SUBAPPLICATION Uebung_001_P (* DigitalInput_I1 auf DigitalOutput_Q1, mit Plug and Socket *)
  (* Standard: 61499-2 *)
  (* Version 1.0, 2023-10-23, franz *)
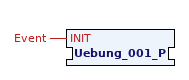
  EVENT_INPUT
    INIT;
  END_EVENT
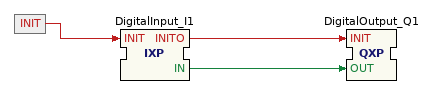
  FBS
    DigitalInput_I1 : IXP;
    DigitalOutput_Q1 : QXP;
  END_FBS
  EVENT_CONNECTIONS
    INIT TO DigitalInput_I1.INIT;
    DigitalInput_I1.INITO TO DigitalOutput_Q1.INIT;
  END_CONNECTIONS
  ADAPTER_CONNECTIONS
    DigitalInput_I1.IN TO DigitalOutput_Q1.OUT;
  END_CONNECTIONS
END_SUBAPPLICATION
